(* IEC 61131-3 sources: volt/packages/volt-lsp-iec/test-corpus/awa-palletizer/Device/Plc Logic/Application/050 Recipe and Machine Parameters, 4 files *)

(* ---- fcCompareStructs.pou ---- *)
FUNCTION fcCompareStructs : BOOL
VAR_INPUT
               PT1 : POINTER TO ARRAY[0..32767] OF BYTE;
               PT2 : POINTER TO ARRAY[0..32767] OF BYTE;
               SIZE1 : INT;
               SIZE2 : INT;
END_VAR
VAR
               START : INT := 0;
               i, j, end : INT;
               firstbyte: BYTE;
END_VAR

%LANGUAGE ST
(*
version 1.1        12. nov. 2009
programmer     hugo
tested by            oscat
https://github.com/simsum/oscat/blob/master/BUFFER_COMP.EXP
*)

(* @END_DECLARATION := '0' *)
(* search for first character match *)

IF size2 <= size1 THEN
	end := size1 - size2;
	firstbyte := PT2^[0];
	FOR i := START TO end DO
		IF PT1^[i] = firstbyte THEN
	    	(* first character matches, now compare rest of array *)
	    	j := 1;
	    	WHILE j < size2 DO
	    	IF pt2^[j] <> pt1^[j+i] THEN EXIT; END_IF;
	    	j := j + 1;
	    	END_WHILE;
	    	(* when J > size2 a match was found return the position i in buffer1 *)
	    	fcCompareStructs := j = size2;
	    	RETURN;
		END_IF;
	END_FOR;
END_IF;
fcCompareStructs := FALSE;

(*
hm 14. nov. 2008           rev 1.0
               original version

hm         12. nov. 2009   rev 1.1
               performance increase

*)

END_FUNCTION

(* ---- fbMachineParManager.pou ---- *)
{attribute 'symbol' := 'none'}
FUNCTION_BLOCK fbMachineParManager
VAR_INPUT
	sDatabaseName		: STRING;	//Database of recipe manager (name)
END_VAR
VAR_OUTPUT
	iNumberOfRecipes	: INT;		//Counted recipes in database
	dwReturnValue		: DWORD;	//Return value of recipe manager
END_VAR
VAR
	RecipeHandler			: RecipeManCommands; //Function to access PLC recipes
	sRecipeLocal			: STRING;          //Used to concat
	// Names
	psNames					: POINTER TO STRING(GLOBAL_CONSTANTS.iSizeRecipesNames);
	// Pointer
	psLocal					: POINTER TO STRING;
	iLoopNames				: INT; //Loop recipe names
	strSearchChar			: STRING;
	iResult					: INT;
	sRecipeName				: STRING;    //Selected recipe (name)
	GetDateAndTime			: rtclk.GetDateAndTime;
	dtDateAndTIme			: DATE_AND_TIME;
	sDateAndTIme			: STRING;
	sDateAndTIme1			: STRING(255);
	sDateAndTIme2			: STRING(255);
	sRecipeNamePar			: STRING(255);
	xSavePar				: BOOL;
	{attribute 'symbol' := 'readwrite'}
	HMI_stRecipeManagercmd	: dutRecipeManagerCmd;
END_VAR

%LANGUAGE ST
GetDateAndTime(
xExecute:= HMI_stRecipeManagercmd.xSave,
dtDateAndTime=> dtDateAndTIme );

sDateAndTIme := TO_STRING(dtDateAndTIme);
sDateAndTIme1:= DELETE(STR:=sDateAndTIme , LEN:=4 , POS:=0 );
sDateAndTIme2:= REPLACE(STR1:= sDateAndTIme1, STR2:='h' , L:=1 , P:=14);
sRecipeNamePar:= REPLACE(STR1:= sDateAndTIme2, STR2:='m' , L:=1 , P:=17);

IF HMI_stRecipeManagercmd.xSave AND GetDateAndTime.xDone THEN
	sRecipeName := sRecipeNamePar;
	xSavePar := TRUE;
	HMI_stRecipeManagercmd.xSave := FALSE;
END_IF

//Get data addresses
psNames := ADR(HMI_stRecipeManagercmd.sRecipeNames);
psLocal := ADR(sRecipeLocal);
//Refresh file buffer
RecipeHandler.ReloadRecipes(sDatabaseName);
//Get recipe count
iNumberOfRecipes := RecipeHandler.GetRecipeCount(sDatabaseName);
//Get saved recipe informations
HMI_stRecipeManagercmd.sRecipeNames:='';
FOR iLoopNames:=0 TO iNumberOfRecipes-1 BY 1 DO
	//Get recipe name
	sRecipeLocal := '';
	RecipeHandler.GetRecipeNames(sDatabaseName, ADR(sRecipeLocal) , 1, iLoopNames);

	//Add recipe name to end of string
	StrConcatA(pstFrom:= psLocal, pstTo:= psNames, iBufferSize:= GLOBAL_CONSTANTS.iSizeRecipesNames);

	//Add seperator to end
	sRecipeLocal := ';';
	StrConcatA(pstFrom:= psLocal, pstTo:= psNames, iBufferSize:= GLOBAL_CONSTANTS.iSizeRecipesNames);
END_FOR

//************************************************************************Load recipe to HMI
IF HMI_stRecipeManagercmd.xLoad THEN
	//Qst_dwReturnValue:=RecipeHandler.LoadAndWriteRecipe(IN_sDatabaseName, sRecipeName);//Load to handler recipe
	dwReturnValue:=RecipeHandler.LoadAndWriteRecipe(sDatabaseName, HMI_stRecipeManagercmd.sSelectedRecipeName);//Load to handler recipe
	IF dwReturnValue = 0 THEN
		HMI_stRecipeManagercmd.sActiveRecipe := HMI_stRecipeManagercmd.sSelectedRecipeName;
	END_IF
	HMI_stRecipeManagercmd.xLoad := FALSE;
END_IF
//************************************************************************Save recipe to database
(*IF HMI_stRecipeManagercmd.xSave THEN
               Qst_dwReturnValue:=RecipeHandler.ReadAndSaveRecipe(IN_sDatabaseName, HMI_stRecipeManagercmd.sActiveRecipe);                   //Save to file
               xSavePar := FALSE;
END_IF*)
//************************************************************************Delete recipe
//More than 0 recipes left
IF HMI_stRecipeManagercmd.xDelete THEN
	dwReturnValue:=RecipeHandler.DeleteRecipe(sDatabaseName, HMI_stRecipeManagercmd.sSelectedRecipeName);               //Remove database link
	IF HMI_stRecipeManagercmd.sActiveRecipe = HMI_stRecipeManagercmd.sSelectedRecipeName THEN
		HMI_stRecipeManagercmd.sActiveRecipe:='';
	END_IF
	HMI_stRecipeManagercmd.xDelete := FALSE;
END_IF
//************************************************************************Save recipe as
IF xSavePar THEN
	strSearchChar:='.';
	iResult:=StrFindA(pst1:=ADR(sRecipeName) , pst2:= ADR(strSearchChar), uiSearchStart:= 0);
	IF iResult <> 0 THEN
		dwReturnValue:=16#7000;
		RETURN;
	END_IF
	dwReturnValue:=RecipeHandler.CreateRecipe(sDatabaseName, sRecipeName); //Create new file and save

	//New recipe OR when recipe already existed
	IF dwReturnValue = 16#4005 OR dwReturnValue = 0 THEN
		dwReturnValue:=RecipeHandler.ReadAndSaveRecipe(sDatabaseName, sRecipeName);  //Create new file and save
	END_IF
	IF dwReturnValue = 0 THEN
		dwReturnValue:=RecipeHandler.LoadAndWriteRecipe(sDatabaseName, sRecipeName);//Load to handler recipe
		dwReturnValue:=SEL(dwReturnValue <> 0, 0, 16#7001);
	END_IF
	IF dwReturnValue = 0 THEN
		HMI_stRecipeManagercmd.sActiveRecipe := sRecipeName;
	END_IF
	xSavePar := FALSE;
END_IF

END_FUNCTION_BLOCK

(* ---- fbRecipeManager.pou ---- *)
{attribute 'symbol' := 'none'}
FUNCTION_BLOCK fbRecipeManager
VAR_INPUT
	sDatabaseName			: STRING;    //Database of recipe manager (name)
END_VAR
VAR_OUTPUT
	iNumberOfRecipes  		: INT;   	//Counted recipes in database
	dwReturnValue     		: DWORD;   	//Return value of recipe manager
	ActiveRecipe        		: dutRecipe;
	{attribute 'symbol' := 'readwrite'}
	xLoadedNewRecipe       	: BOOL;
	{attribute 'symbol' := 'readwrite'}
	xRcpVisuPlcAreEqual		: BOOL;
END_VAR
VAR
	NewRecipe 			: dutRecipe;  //Initial recipe values
	RecipeHandler             	: RecipeManCommands; 	//Function to access PLC recipes
	sRecipeLocal                : STRING;           	//Used to concat
	psNames            			: POINTER TO STRING(gc_iSizeRecipesNames);
	psLocal       				: POINTER TO STRING;
	iLoopNames         			: INT;    //Loop recipe names
	strSearchChar          		: STRING;
	iResult                 	: INT;
	sRecipNameTemp           	: STRING;

	F_TRIG_Save	: F_TRIG;
	F_TRIG_Load	: F_TRIG;
	xSaveStarted:BOOL;
END_VAR
VAR RETAIN PERSISTENT

	//HMI
	{attribute 'symbol' := 'readwrite'}
	HMI_stRecipeVisu         	: dutRecipe;
END_VAR
VAR
	{attribute 'symbol' := 'readwrite'}
	HMI_stRecipeManagercmd  	: dutRecipeManagerCmd;
END_VAR
VAR CONSTANT
	gc_iSizeRecipesNames    	: INT := 16384;
END_VAR

%LANGUAGE ST

xLoadedNewRecipe := FALSE;

//Get data addresses
psNames := ADR(HMI_stRecipeManagercmd.sRecipeNames);
psLocal := ADR(sRecipeLocal);

//Refresh file buffer
RecipeHandler.ReloadRecipes(sDatabaseName);

//Get recipe count
iNumberOfRecipes := RecipeHandler.GetRecipeCount(sDatabaseName);

//Get saved recipe informations
HMI_stRecipeManagercmd.sRecipeNames:='';
FOR iLoopNames:=0 TO iNumberOfRecipes-1 BY 1 DO
    //Get recipe name
    sRecipeLocal := '';
    RecipeHandler.GetRecipeNames(sDatabaseName, ADR(sRecipeLocal) , 1, iLoopNames);

    //Add recipe name to end of string
    StrConcatA(pstFrom:= psLocal, pstTo:= psNames, iBufferSize:= gc_iSizeRecipesNames);

    //Add seperator to end
    sRecipeLocal := ';';
    StrConcatA(pstFrom:= psLocal, pstTo:= psNames, iBufferSize:= gc_iSizeRecipesNames);
END_FOR

IF HMI_stRecipeManagercmd.xLoad THEN
	dwReturnValue:=RecipeHandler.LoadAndWriteRecipe(sDatabaseName, HMI_stRecipeManagercmd.sSelectedRecipeName);//Load to handler recipe
	IF dwReturnValue = 0 THEN
		ActiveRecipe:=HMI_stRecipeVisu;
		HMI_stRecipeManagercmd.sActiveRecipe := HMI_stRecipeManagercmd.sSelectedRecipeName;
	END_IF
	xLoadedNewRecipe := TRUE;
	HMI_stRecipeManagercmd.xLoad:=FALSE;
END_IF

IF HMI_stRecipeManagercmd.xNew THEN
	sRecipNameTemp := HMI_stRecipeVisu.sRecipeName;
	HMI_stRecipeVisu:= NewRecipe; // to set the initial recipe values
	HMI_stRecipeVisu.sRecipeName:= sRecipNameTemp;
	strSearchChar:='.';
	dwReturnValue:=INT_TO_DWORD(StrFindA(pst1:=ADR(HMI_stRecipeVisu.sRecipeName) , pst2:= ADR(strSearchChar), uiSearchStart:= 0));
	IF dwReturnValue = 0 THEN
		dwReturnValue:=RecipeHandler.CreateRecipe(sDatabaseName, HMI_stRecipeVisu.sRecipeName);
		HMI_stRecipeManagercmd.sSelectedRecipeName := HMI_stRecipeVisu.sRecipeName;
	ELSE
		dwReturnValue:=16#7000;
	END_IF
	HMI_stRecipeManagercmd.xNew := FALSE;
END_IF

IF HMI_stRecipeManagercmd.xEdit THEN
	dwReturnValue:=RecipeHandler.LoadAndWriteRecipe(sDatabaseName, HMI_stRecipeManagercmd.sSelectedRecipeName);//Load to handler recipe
	HMI_stRecipeManagercmd.xEdit:=FALSE;
END_IF

IF HMI_stRecipeManagercmd.xSave THEN
	dwReturnValue:=RecipeHandler.ReadAndSaveRecipe(sDatabaseName, HMI_stRecipeVisu.sRecipeName); //Create new file and save
	HMI_stRecipeManagercmd.xSave := FALSE;
END_IF

IF HMI_stRecipeManagercmd.xCopy THEN
	 sRecipNameTemp:=HMI_stRecipeVisu.sRecipeName;
	dwReturnValue:=RecipeHandler.LoadAndWriteRecipe(sDatabaseName, HMI_stRecipeManagercmd.sSelectedRecipeName);
	HMI_stRecipeVisu.sRecipeName:=sRecipNameTemp;
	strSearchChar:='.';
	dwReturnValue:=INT_TO_DWORD(StrFindA(pst1:=ADR(HMI_stRecipeVisu.sRecipeName) , pst2:= ADR(strSearchChar), uiSearchStart:= 0));
	IF dwReturnValue = 0 THEN
		dwReturnValue:=RecipeHandler.CreateRecipe(sDatabaseName, HMI_stRecipeVisu.sRecipeName);
		HMI_stRecipeManagercmd.sSelectedRecipeName := HMI_stRecipeVisu.sRecipeName;
    ELSE
          dwReturnValue:=16#7000;
    END_IF
    HMI_stRecipeManagercmd.xCopy := FALSE;
END_IF

IF HMI_stRecipeManagercmd.xDelete THEN
	dwReturnValue:=RecipeHandler.DeleteRecipe(sDatabaseName, HMI_stRecipeManagercmd.sSelectedRecipeName); //Remove database link
	HMI_stRecipeManagercmd.xDelete := FALSE;
END_IF

IF HMI_stRecipeManagercmd.xUpdate THEN
	HMI_stRecipeVisu:=ActiveRecipe;
	dwReturnValue:=RecipeHandler.ReadAndSaveRecipe(sDatabaseName, HMI_stRecipeVisu.sRecipeName); //Create new file and save
	HMI_stRecipeManagercmd.xUpdate := FALSE;
END_IF

IF HMI_stRecipeManagercmd.xSaveAndLoad THEN
	IF F_TRIG_Save.Q THEN
		HMI_stRecipeManagercmd.xLoad := TRUE;
	END_IF
	IF F_TRIG_Load.Q THEN
		HMI_stRecipeManagercmd.xSaveAndLoad := FALSE;
	END_IF

	IF NOT(HMI_stRecipeManagercmd.xsave) AND NOT(xSaveStarted) THEN
		HMI_stRecipeManagercmd.xsave := TRUE;
		xSaveStarted:= TRUE;
	END_IF
ELSE
	xSaveStarted := FALSE;
END_IF

F_TRIG_Save(CLK := HMI_stRecipeManagercmd.xsave);
F_TRIG_Load(CLK := HMI_stRecipeManagercmd.xLoad);

HMI_stRecipeManagercmd.xRcpVisuPlcAreEqual := fcCompareStructs(PT1:=ADR(ActiveRecipe) ,PT2:=ADR(HMI_stRecipeVisu), SIZE1:=TO_INT(SIZEOF(ActiveRecipe)), SIZE2:=TO_INT(SIZEOF(HMI_stRecipeVisu)));

END_FUNCTION_BLOCK

(* ---- pgRecipeHandler.pou ---- *)
{attribute 'symbol' := 'none'}
PROGRAM pgRecipeHandler
VAR
	{attribute 'symbol' := 'readwrite'}
	RecipeManager				: fbRecipeManager;
	{attribute 'symbol' := 'readwrite'}
	MachineParManager				: fbMachineParManager;
END_VAR
VAR_OUTPUT
	iNumberOfMachinePar  		: INT;   	//Counted recipes in database
	iNumberOfRecipes  		: INT;   	//Counted recipes in database
	ActiveRecipe        	: dutRecipe;
	xLoadedNewRecipe       	: BOOL;
	xRcpVisuPlcAreEqual		: BOOL;
END_VAR
VAR
	dwRecipeReturnValue		: DWORD;	//Return value of recipe manager
	// Return value of machine par manager
	dwMachineParReturnValue: DWORD;
END_VAR

%LANGUAGE FBD
%NETWORK
RecipeManager(EN := TRUE, sDatabaseName := 'Recipes', iNumberOfRecipes => iNumberOfRecipes, dwReturnValue => dwRecipeReturnValue, ActiveRecipe => ActiveRecipe, xLoadedNewRecipe => xLoadedNewRecipe, xRcpVisuPlcAreEqual => xRcpVisuPlcAreEqual);
%NETWORK
MachineParManager(EN := TRUE, sDatabaseName := 'MachinePar', iNumberOfRecipes => iNumberOfMachinePar, dwReturnValue => dwMachineParReturnValue);

END_PROGRAM
